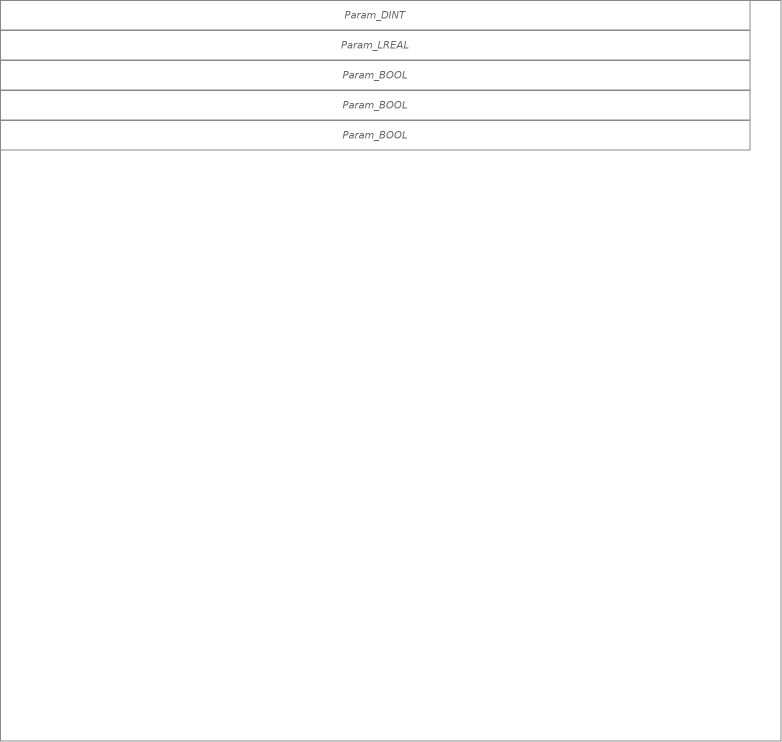
VISUALIZATION Visu_Mparam_Extruder  // 782x742
    Frame (0,30 750x30)
        shows Param_LREAL(nIdx := 3)
    Frame (0,90 750x30)
        shows Param_BOOL(nIdx := 8)
    Frame (0,60 750x30)
        shows Param_BOOL(nIdx := 2)
    Frame (0,0 750x30)
        shows Param_DINT(nIdx := 3)
    Frame (0,120 750x30)
        shows Param_BOOL(nIdx := 14)
    Rectangle (30,710 750x30)
END_VISUALIZATION

(* stored: Version 1.1.0.1, ProductVersion 3.1.4024.12
   Visu Visu_Mparam_Extruder: Id {c3fa1c15-09d5-44f0-9fed-7e2deb5b3cda} *)
